(* CODESYS project Mudpi.library
   Company: ESO
   DefaultNamespace: ESO.MUDPI
   Title: ESO MUDPI Library
   Description: This library provides functionality to pack/unpack frames in the MUDPI format (Multicast UDP interface). The data format for MUDPI is described in the document "ESO-302020 - MUDPI Format".
   Placeholder: ESO MUDPI Library
   Author: Jakob Sagatowski
   Version: 1.0.1.0

Project tree, tasks and I/O mapping:
  libraries: Tc2_Standard, * (Beckhoff Automation GmbH); Tc2_System, * (Beckhoff Automation GmbH); Tc2_Utilities, * (Beckhoff Automation GmbH); Tc3_Module, * (Beckhoff Automation GmbH); TcUnit, * (www.tcunit.org)
  DUTs/
    data type ST_MudpiDataType
    data type ST_MudpiHeaderType
  GVLs/
    global variables GVL
  POUs/
    function block FB_MudpiPacket [ST]: CalculateChecksum, Data, FB_init, GetApplicationTag, GetChecksum, GetComponentId, GetFrameId, GetMaxPayloadSize, GetNumFrames, GetPayload, GetPayloadSize, GetSampleId, GetTimestamp, GetTopicId, GetVersion, IncreaseSampleId, Initialize, SetApplicationTag, SetChecksum, SetComponentId, SetFrameId, SetNumFrames, SetPayload, SetPayloadSize, SetSampleId, SetTimestamp, SetTopicId, SetVersion, Size, VerifyChecksum, VerifyPacket
  Test/
    function block FB_MudpiPacket_Test [ST]: TestChecksumCalculation, TestChecksumCalculationForPayload, TestCorrectSizeOfMudpiPacketWithAndWithoutPayload, TestPacketIntegrityMethod, TestPayloadDataSize, TestSampleIdIncreaseCorrectly, TestSerializationOfMudpiPacket, TestSetAndGetMethodForTimestamp, TestStoreAndRetrieveOfConstructorValues, TestValidAndInvalidMudpiPacketInitialization
    program PRG_TEST [ST]
  Version/
    global variables Global_Version
  VISUs/
*)

// DUTs/ST_MudpiDataType
{attribute 'pack_mode' := '1'} 
TYPE ST_MudpiDataType :
STRUCT
    header : ST_MudpiHeaderType;
    data : ARRAY[0..(GVL.MUDPI_PAYLOAD_SIZE - 1)] OF BYTE;
END_STRUCT
END_TYPE

// DUTs/ST_MudpiHeaderType
(**
 * TYPEDEF for a MUDPI header. The structure is as follows:
 *
 * UDINT TopicId         // Unique identifier of data topic
 * UINT  ComponentId     // Unique identifier of the sender
 * UINT  ApplicationTag  // For application use (not used by MUDPI)
 * UINT  Reserved1       // Reserved for future use
 * UINT  Version         // MUDPI version identifier
 * UDINT SampleId        // Rolling sample identifier (thus not unique, rather an incrementing number), incremented for each new sample
 * ULINT Timestamp       // Seconds since UNIX Epoch, following TAI time line
 * UINT  FrameId         // Frame counter for multi‐frame transmissions (starting from 1)
 * UINT  NumFrames       // Number of frames in a multi‐part message
 * UINT  PayloadSize     // Size in bytes of the payload
 * UINT  Reserved2       // Reserved for future use
 *)
 
{attribute 'pack_mode' := '1'} 
TYPE ST_MudpiHeaderType :
STRUCT
    topicId : UDINT;
    componentId : UINT;
    applicationTag : UINT;
    reserved1 : UINT;
    version : UINT;
    sampleId : UDINT;
    timestamp : ULINT;
    frameId : UINT;
    numFrames : UINT;
    payloadSize : UINT;
    reserved2 : UINT;
END_STRUCT
END_TYPE

// GVLs/GVL
(*
    MUDPI constants
*)
 
{attribute 'qualified_only'}
VAR_GLOBAL CONSTANT
    IEEE802_3_PAYLOAD_SIZE : UINT := 1500; (* = IEEE802.3 ethernet basic frame payload *)
    IPV4_HEADER_SIZE : UINT := 20;
    UDP_HEADER_SIZE : UINT := 8;
    MUDPI_PAYLOAD_SIZE : UINT := IEEE802_3_PAYLOAD_SIZE - IPV4_HEADER_SIZE - UDP_HEADER_SIZE  - SIZEOF(ST_MudpiHeaderType);
    MUDPI_VERSION : UINT := 1;
END_VAR

// Version/Global_Version
{attribute 'TcGenerated'}
{attribute 'no-analysis'}
{attribute 'linkalways'}
// This function has been automatically generated from the project information.
VAR_GLOBAL CONSTANT
	{attribute 'const_non_replaced'}
	stLibVersion_ESO_MUDPI_Library : ST_LibVersion := (iMajor := 1, iMinor := 0, iBuild := 1, iRevision := 0, sVersion := '1.0.1.0');
END_VAR

// POUs/FB_MudpiPacket
(*
    This function block gives a definition of a MUDPI packet. The MUDPI format is described in ESO document
    ESO-302020.

    As it's not possible to have more than one "constructor" in IEC61131-3, the packet is initialized in a different
    way depending on whether it's going to be used for transmission or reception.
    For transmission:
    - Just create an instance of the function block by supplying the necessary parameters to the constructor.
      All the other variables can be changed by the applicable set-methods.
    For reception:
    - Create an instance of the function block by supplying the necessary parameters to the constructor. The parameters
      can be dummy as these are going to be overwritten. Once the object is instantiated, call the method
      Initialize() on it and supply the input parameters for the data.
*)
FUNCTION_BLOCK FB_MudpiPacket
VAR
    mData : ST_MudpiDataType;
END_VAR

(*
    Calculates 16-bit UDP checksum (zero indicates no checksum).

    All 16-bit words are summed using one's complement arithmetic. Add the 16-bit values up. Each time a
    carry-out (17th bit) is produced, swing that bit around and add it back into the least significant bit.
    The sum is then one's complemented to yield the value of the UDP checksum field. If the computed
    checksum is zero, it is transmitted as all ones (the equivalent in one's complement arithmetic).
    An all zero transmitted checksum value means that the transmitter generated no checksum (for debugging
    or for higher level protocols that don't care).

*)
METHOD PUBLIC CalculateChecksum : UINT
VAR
    packetSize : UINT;
    dataPointer : POINTER TO UINT;
    dataPointerSmall : POINTER TO USINT;

    sum : UDINT := 0;
    returnValue : UINT;
END_VAR
packetSize := GetPayloadSize();
packetSize := packetSize + SIZEOF(ST_MudpiHeaderType);

dataPointer := ADR(mData.header);

// Calculate 1's complement sum of the data
WHILE (packetSize > 1) DO
    sum := sum + dataPointer^;
    dataPointer := dataPointer + SIZEOF(UINT);

    IF ((sum AND 16#80000000) = 10#1) THEN
        sum := (sum AND 16#FFFF) + (SHR(sum, 16));
    END_IF
    packetSize := packetSize - SIZEOF(UINT);
END_WHILE

IF ((packetSize AND 10#1) <> 10#0) THEN
    dataPointerSmall := dataPointer;
    sum := sum + dataPointerSmall^;
END_IF

// Add carry-over
WHILE (SHR(sum, 16)) > 10#0 DO
    sum := (sum AND 16#FFFF) + (SHR(sum, 16));
END_WHILE
returnValue := UDINT_TO_UINT(NOT sum);

IF returnValue = 0 THEN
    returnValue := NOT returnValue;
END_IF

CalculateChecksum := returnValue;
END_METHOD

(*
    Returns a pointer to the packet, be aware that the contents are big-endian!
*)
METHOD PUBLIC Data : POINTER TO BYTE
VAR
    checksum : UINT;
END_VAR
checksum := CalculateChecksum();
SetChecksum(checksum := checksum);

Data := ADR(mData);
END_METHOD

METHOD FB_init : BOOL
VAR_INPUT
    bInitRetains : BOOL; // if TRUE, the retain variables are initialized (warm start / cold start)
    bInCopyCode : BOOL;  // if TRUE, the instance afterwards gets moved into the copy code (online change)
    topicId : UDINT;
    componentId : UINT;
END_VAR
SetVersion(Version := GVL.MUDPI_VERSION);
SetFrameId(FrameId := 1);
SetNumFrames(NumFrames := 1);
SetTopicId(TopicId := topicId);
SetComponentId(ComponentId := componentId);
END_METHOD

METHOD PUBLIC GetApplicationTag : UINT
GetApplicationTag := WORD_TO_UINT(Tc2_Utilities.BE16_TO_HOST(in := UINT_TO_WORD(mData.header.applicationTag)));
END_METHOD

METHOD PUBLIC GetChecksum : UINT
VAR
    payloadSize : UINT;
    checksum : UINT;
END_VAR
payloadSize := GetPayloadSize();
Tc2_System.MEMCPY(destAddr := ADR(checksum), srcAddr := ADR(mData.data[payloadSize]), n := SIZEOF(UINT));
GetChecksum := checksum;
END_METHOD

METHOD PUBLIC GetComponentId : UINT
GetComponentId := WORD_TO_UINT(Tc2_Utilities.BE16_TO_HOST(in := UINT_TO_WORD(mData.header.componentId)));
END_METHOD

METHOD PUBLIC GetFrameId : UINT
GetFrameId := WORD_TO_UINT(Tc2_Utilities.BE16_TO_HOST(in := UINT_TO_WORD(mData.header.frameId)));
END_METHOD

(*
    Returns maximum payload size.
*)
METHOD PUBLIC GetMaxPayloadSize : UINT
GetMaxPayloadSize := GVL.MUDPI_PAYLOAD_SIZE;
END_METHOD

METHOD PUBLIC GetNumFrames : UINT
GetNumFrames := WORD_TO_UINT(Tc2_Utilities.BE16_TO_HOST(in := UINT_TO_WORD(mData.header.numFrames)));
END_METHOD

METHOD PUBLIC GetPayload : POINTER TO BYTE
GetPayload := ADR(mData.data[0]);
END_METHOD

METHOD PUBLIC GetPayloadSize : UINT
GetPayloadSize := WORD_TO_UINT(Tc2_Utilities.BE16_TO_HOST(in := UINT_TO_WORD(mData.header.payloadSize)));
END_METHOD

METHOD PUBLIC GetSampleId : UDINT
GetSampleId := DWORD_TO_UDINT(Tc2_Utilities.BE32_TO_HOST(in := UDINT_TO_DWORD(mData.header.sampleId)));
END_METHOD

(*
    This method returns the timestamp of a MUDPI packet.
    The timestamp is in seconds since UNIX Epoch, following TAI time line.
 *)
METHOD PUBLIC GetTimestamp : LREAL
VAR
    timestampLocal : LREAL;
    tmp : ULINT;
END_VAR
tmp := LWORD_TO_ULINT(Tc2_Utilities.BE64_TO_HOSTEX(in := ULINT_TO_LWORD(mdata.header.timestamp)));
Tc2_System.MEMCPY(destAddr := ADR(timestampLocal), srcAddr := ADR(tmp), n := SIZEOF(LREAL));

GetTimestamp := TimestampLocal;
END_METHOD

METHOD PUBLIC GetTopicId : UDINT
GetTopicId := DWORD_TO_UDINT(Tc2_Utilities.BE32_TO_HOST(in := UDINT_TO_DWORD(mData.header.topicId)));
END_METHOD

METHOD PUBLIC GetVersion : UINT
GetVersion := WORD_TO_UINT(Tc2_Utilities.BE16_TO_HOST(in := UINT_TO_WORD(mData.header.version)));
END_METHOD

(*
    This method increases the sample ID of the MUDPI packet.
*)
METHOD PUBLIC IncreaseSampleId
VAR
    mySampleId : UDINT;
END_VAR
mySampleId := GetSampleId();
mySampleId := mySampleId + 1;
SetSampleId(SampleId := mySampleId);
END_METHOD

(*
    This method create the MUDPI structure from a stream of bytes.
    TRUE = Creation successful, FALSE = Input data too large for MUDPI packet
*)
METHOD PUBLIC Initialize : BOOL
VAR_INPUT
    inputData : POINTER TO BYTE;
    size : UINT;
END_VAR
VAR
    sizeTmp : UINT;
END_VAR
sizeTmp := GVL.MUDPI_PAYLOAD_SIZE + SIZEOF(ST_MudpiHeaderType);

IF (size <= sizeTmp) THEN
    Tc2_System.MEMCPY(destAddr := ADR(mData), srcAddr := inputData, n := size);
    Initialize := TRUE;
ELSE
    Initialize := FALSE;
END_IF
END_METHOD

METHOD PUBLIC SetApplicationTag
VAR_INPUT
    ApplicationTag : UINT;
END_VAR
mData.header.applicationTag := WORD_TO_UINT(Tc2_Utilities.HOST_TO_BE16(in := UINT_TO_WORD(ApplicationTag)));
END_METHOD

METHOD PUBLIC SetChecksum
VAR_INPUT
    checksum : UINT;
END_VAR
VAR
    payloadSize : UINT;
END_VAR
payloadSize := GetPayloadSize();
Tc2_System.MEMCPY(destAddr := ADR(mData.data[payloadSize]), srcAddr := ADR(checksum), SIZEOF(checksum));
END_METHOD

METHOD PUBLIC SetComponentId
VAR_INPUT
    ComponentId : UINT;
END_VAR
mData.header.componentId := WORD_TO_UINT(Tc2_Utilities.HOST_TO_BE16(in := UINT_TO_WORD(ComponentId)));
END_METHOD

METHOD PUBLIC SetFrameId
VAR_INPUT
    FrameId : UINT;
END_VAR
mData.header.frameId := WORD_TO_UINT(Tc2_Utilities.HOST_TO_BE16(in := UINT_TO_WORD(FrameId)));
END_METHOD

METHOD PUBLIC SetNumFrames
VAR_INPUT
    NumFrames : UINT;
END_VAR
mData.header.numFrames := WORD_TO_UINT(Tc2_Utilities.HOST_TO_BE16(in := UINT_TO_WORD(NumFrames)));
END_METHOD

(*
    This method sets the payload of a MUDPI packet.

    payload: Pointer to any data.
    payloadSize: Size of payload data in bytes.

    Return value: TRUE = Payload set successfully, FALSE = Not possible to set payload. Payload too large for MUDPI packet.
 *)
METHOD PUBLIC SetPayload : BOOL
VAR_INPUT
    payload : POINTER TO BYTE;
    payloadSize : UINT;
END_VAR
IF (payloadSize > (GVL.MUDPI_PAYLOAD_SIZE - SIZEOF(UINT))) THEN // SIZEOF(UINT) = Checksum
    SetPayload := FALSE;
ELSE
    IF (payloadSize > 0) THEN
        SetPayloadSize(payloadSize);
        Tc2_System.MEMCPY(destAddr := ADR(mData.data[0]), srcAddr := payload, n := payloadSize);
    END_IF
    SetPayload := TRUE;
END_IF
END_METHOD

METHOD PUBLIC SetPayloadSize
VAR_INPUT
    PayloadSize : UINT;
END_VAR
mData.header.payloadSize := WORD_TO_UINT(Tc2_Utilities.HOST_TO_BE16(in := UINT_TO_WORD(PayloadSize)));
END_METHOD

METHOD PUBLIC SetSampleId
VAR_INPUT
    SampleId : UDINT;
END_VAR
mData.header.sampleId := DWORD_TO_UDINT(Tc2_Utilities.HOST_TO_BE32(in := UDINT_TO_DWORD(SampleId)));
END_METHOD

(*
    This method sets the timestamp of a MUDPI packet.
    The timestamp is in seconds since UNIX Epoch, following TAI time line.
 *)
METHOD PUBLIC SetTimestamp
VAR_INPUT
    Timestamp : LREAL;
END_VAR
VAR
    TimestampLocal : ULINT;
END_VAR
Tc2_System.MEMCPY(destAddr := ADR(TimestampLocal), srcAddr := ADR(Timestamp), n := SIZEOF(LREAL));
mData.header.timestamp := LWORD_TO_ULINT(Tc2_Utilities.HOST_TO_BE64EX(in := ULINT_TO_LWORD(TimestampLocal)));
END_METHOD

METHOD PUBLIC SetTopicId
VAR_INPUT
    TopicId : UDINT;
END_VAR
mData.header.topicId := DWORD_TO_UDINT(Tc2_Utilities.HOST_TO_BE32(in := UDINT_TO_DWORD(TopicId)));
END_METHOD

METHOD PUBLIC SetVersion
VAR_INPUT
    Version : UINT;
END_VAR
mData.header.version := WORD_TO_UINT(Tc2_Utilities.HOST_TO_BE16(in := UINT_TO_WORD(Version)));
END_METHOD

(*
    This method returns the size of the MUDPI packet in bytes.
    The return value is the size of the packet in bytes, i.e. MUDPI header + payload + checksum.
 *)
METHOD PUBLIC Size : UINT
VAR
    payloadSize : UINT;
    sizeOfMudpiHeader : UINT := SIZEOF(ST_MudpiHeaderType);
    sizeOfChecksum : UINT := SIZEOF(UINT);
END_VAR
payloadSize := GetPayloadSize();
Size := payloadSize + sizeOfMudpiHeader + sizeOfChecksum;
END_METHOD

(*
    This method verifies, if the checksum of a MUDPI packet is correct.
    TRUE = Checksum does match the content of the packet, FALSE = checksum does not match.
*)
METHOD PUBLIC VerifyChecksum : BOOL
VAR
    checksum1 : UINT;
    checksum2 : UINT;
END_VAR
checksum1 := GetChecksum();
checksum2 := CalculateChecksum();

// The MUDPI standard allows to omit the checksum calculation
IF ((checksum1 = 0) OR (checksum2 = 0)) THEN
    VerifyChecksum := TRUE;
ELSE
    VerifyChecksum := (checksum1 = checksum2);
END_IF
END_METHOD

(*
    This method verifies, if the internal structure of a MUDPI packet is correct.
    TRUE = internal structure of packet is correct, FALSE = internal structure of packet is not correct
*)
METHOD PUBLIC VerifyPacket : BOOL
VAR
    version : UINT;
    frameId : UINT;
    numFrames : UINT;
    topicId : UDINT;
    componentId : UINT;
    checksumCorrect : BOOL;
    packetCorrect : BOOL;
END_VAR
version := GetVersion();
frameId := GetFrameId();
numFrames := GetNumFrames();
topicId := GetTopicId();
componentId := GetComponentId();

checksumCorrect := VerifyChecksum();
packetCorrect := (version = GVL.MUDPI_VERSION) AND (frameId <= numFrames) AND (topicId <> 0) AND (componentId <> 0);

VerifyPacket := (checksumCorrect AND packetCorrect);
END_METHOD

END_FUNCTION_BLOCK

// Test/FB_MudpiPacket_Test
(*
    This is the test-FB for FB_MudpiPacket
*)
{attribute 'call_after_init'}
FUNCTION_BLOCK FB_MudpiPacket_Test EXTENDS TcUnit.FB_TestSuite
VAR CONSTANT
    cTopicId : UDINT := 10;
    cComponentId : UINT := 500;
END_VAR

TestStoreAndRetrieveOfConstructorValues();
TestCorrectSizeOfMudpiPacketWithAndWithoutPayload();
TestPayloadDataSize();
TestChecksumCalculationForPayload();
TestSampleIdIncreaseCorrectly();
TestPacketIntegrityMethod();
TestSerializationOfMudpiPacket();
TestValidAndInvalidMudpiPacketInitialization();
TestSetAndGetMethodForTimestamp();
TestChecksumCalculation();

(*
    Test checksum calculation for given header

    The header should be according to:
    - TopicId = 500
    - ComponentId = 10
    - ApplicationTag = 300
    - SampleId = 422
    - NumFrames = 212
    - Version = 1
    - Timestamp = 0
    - FrameId = 1
    - No Payload
*)
METHOD PRIVATE TestChecksumCalculation
VAR
    // Construct MUDPI packet
    packet : FB_MudpiPacket(topicId := 500, componentId := 10);

    checksum : UINT;
END_VAR
TEST('TestChecksumCalculation');

packet.SetApplicationTag(ApplicationTag := 300);
packet.SetSampleId(SampleId := 422);
packet.SetNumFrames(NumFrames := 212);
packet.SetVersion(Version := 1);
packet.SetTimeStamp(Timestamp := 0.0);
packet.SetFrameId(FrameId := 1);

checksum := packet.CalculateChecksum();

AssertEquals_UINT(Expected := Tc2_Utilities.HOST_TO_BE16(16#FA59),
                  Actual := checksum,
                  Message := 'Calculated checksum is not correct');

TEST_FINISHED();
END_METHOD

(*
    Test checksum calculation for a given payload, and for empty payload data.
*)
METHOD PRIVATE TestChecksumCalculationForPayload
VAR
    // Construct MUDPI packet
    packet : FB_MudpiPacket(topicId := cTopicId, componentId := cComponentId);

    payloadParam : STRING := 'This is a payload';
    checkChecksum1 : BOOL;

    checksum1 : UINT;
    checksum2 : UINT;
END_VAR
TEST('TestChecksumCalculationForPayload');

packet.SetPayload(payload := ADR(payloadParam),
                  payloadSize := SIZEOF(payloadParam));

// Invoke calculation of checksum
packet.Data();

// Verify, if checksum was calculated correctly
checkChecksum1 := packet.VerifyChecksum();

AssertTrue(Condition := checkChecksum1,
           Message := 'Checksum not calculated correctly');

// Calculate checksum, and verify if identical to setting in MUDPI packet
checksum1 := packet.CalculateChecksum();
checksum2 := packet.GetChecksum();

AssertEquals_UINT(Expected := checksum1,
                  Actual := checksum2,
                  Message := 'Calculated checksum not identical with the one in MUDPI packet');

TEST_FINISHED();
END_METHOD

(*
    Test correct return value of size() method with and without payload.
    Test correct return value of getMaxPayloadSize
*)
METHOD PRIVATE TestCorrectSizeOfMudpiPacketWithAndWithoutPayload
VAR
    // Construct MUDPI packet
    packet : FB_MudpiPacket(topicId := cTopicId, componentId := cComponentId);

    sizeHeader : UINT;
    sizeReturned : UINT;
    sizeCorrect : BOOL;

    payloadSize : UINT;
    maxPayloadSize : UINT;

    payload : STRING(9) := '123456789'; // 10 bytes (including the null-character)
END_VAR
TEST('TestCorrectSizeOfMudpiPacketWithAndWithoutPayload');

// Test correct size of MUDPI header
sizeHeader := SIZEOF(ST_MudpiHeaderType);
sizeReturned := packet.Size() - SIZEOF(UINT); // Checksum

AssertEquals_UINT(Expected := sizeHeader,
                  Actual := sizeReturned,
                  Message := 'Size of MUDPI header not correct');

// Test correct size of MUDPI packet with payload of 10 bytes (+checksum internally)
packet.SetPayload(payload := ADR(payload),
                  payloadSize := SIZEOF(payload));
payloadSize := packet.GetPayloadSize();
sizeReturned := packet.Size();
AssertEquals_UINT(Expected := SIZEOF(payload),
                  Actual := payloadSize,
                  Message := 'Size of MUDPI payload not correct');
AssertEquals_UINT(Expected := (sizeHeader + SIZEOF(payload) + SIZEOF(UINT)), // SIZEOF(UINT) = Checksum
                  Actual := sizeReturned,
                  Message := 'Total size of MUDPI-packet including payload not correct');

// Test correct return value of getMaxPayloadSize
maxPayloadSize := packet.GetMaxPayloadSize();
AssertEquals_UINT(Expected := GVL.MUDPI_PAYLOAD_SIZE,
                  Actual := maxPayloadSize,
                  Message := 'The returned value for maximum payload size for the MUDPI packet is not correct');

TEST_FINISHED();
END_METHOD

METHOD PRIVATE TestPacketIntegrityMethod
VAR
    // Construct MUDPI packet
    packet : FB_MudpiPacket(topicId := cTopicId, componentId := cComponentId);
END_VAR
TEST('TestPacketIntegrityMethod');

packet.IncreaseSampleId();

AssertTrue(Condition := packet.VerifyPacket(),
           Message := 'MUDPI packet integrity failed');

TEST_FINISHED();
END_METHOD

(*
    Test setting and retrieving of payload data.
    Test the correct return value for the payload length for packets with and without payload data.
*)
METHOD PRIVATE TestPayloadDataSize
VAR
    // Construct MUDPI packet
    packet : FB_MudpiPacket(topicId := cTopicId, componentId := cComponentId);

    emptyPayloadSize : UINT;
    newPayloadSize : UINT;

    payload : STRING(17) := 'This is a payload'; // 18 bytes (including the null-character)
END_VAR
TEST('TestPayloadDataSize');

// Verify that the payload is empty
emptyPayloadSize := packet.GetPayloadSize();

AssertEquals_UDINT(Expected := 0,
                   Actual := emptyPayloadSize,
                   Message := 'MUDPI payload size is not zero');

// Set a new payload, and verify correct length
packet.SetPayload(payload := ADR(payload),
                  payloadSize := SIZEOF(payload));

newPayloadSize := packet.GetPayloadSize();

AssertEquals_UDINT(Expected := SIZEOF(payload),
                   Actual := newPayloadSize,
                   Message := 'MUDPI payload size is not correct');

TEST_FINISHED();
END_METHOD

(*
    Test, if the sampleId is increased correctly.
*)
METHOD TestSampleIdIncreaseCorrectly
VAR
    // Construct MUDPI packet
    packet : FB_MudpiPacket(topicId := cTopicId, componentId := cComponentId);

    firstSampleId : UDINT;
    secondSampleId : UDINT;
END_VAR
TEST('TestSampleIdIncreaseCorrectly');

// Get initial and increased sampleId
firstSampleId := packet.GetSampleId();
packet.IncreaseSampleId();
secondSampleId := packet.GetSampleId();

AssertEquals_UDINT(Expected := 0,
                   Actual := firstSampleId,
                   Message := 'First Sample-ID not correct');

AssertEquals_UDINT(Expected := 1,
                   Actual := secondSampleId,
                   Message := 'Second Sample-ID not correct');

TEST_FINISHED();
END_METHOD

(*
    Test correct serialization of the MUDPI packet.
*)
METHOD PRIVATE TestSerializationOfMudpiPacket
VAR
    // Construct MUDPI packet
    packet : FB_MudpiPacket(topicId := cTopicId, componentId := cComponentId);

    aByteArray : ARRAY[0..3] OF BYTE;
    serializedData : POINTER TO BYTE;
END_VAR
TEST('TestSerializationOfMudpiPacket');

(* We expect big-endian format, i.e. the bytes in the following order:
    Topic-ID: 0x11, 0x22, 0x33, 0x44
    Component-ID: 0x55, 0x66
    Application-tag: 0x77, 0x88
    Reserved: 0x00, 0x00
    Version: 0x99, 0xAA
    Sample-ID: 0xBB, 0xCC, 0xDD, 0xEE
    Timestamp: 0x40, 0x93, 0x4A, 0x00, 0x00, 0x00, 0x00, 0x00
    Frame-ID: 0x88, 0x99
    NumFrames: 0xAA, 0xBB
    Payload size: 0x01, 0xFF
    Reserved: 0x00, 0x00
*)
packet.SetTopicId(16#11223344);
packet.SetComponentId(16#5566);
packet.SetApplicationTag(16#7788);
packet.SetVersion(16#99AA);
packet.SetSampleId(16#BBCCDDEE);
packet.SetTimeStamp(1234.5); // 1234.5 = 16#40934A0000000000
packet.SetFrameId(16#8899);
packet.SetNumFrames(16#AABB);
packet.SetPayloadSize(16#01FF);

serializedData := packet.Data();
AssertEquals_BYTE(Expected := 16#11,
                  Actual := serializedData[0],
                  Message := 'Byte 0 is not correctly serialized');
AssertEquals_BYTE(Expected := 16#22,
                  Actual := serializedData[1],
                  Message := 'Byte 1 is not correctly serialized');
AssertEquals_BYTE(Expected := 16#33,
                  Actual := serializedData[2],
                  Message := 'Byte 2 is not correctly serialized');
AssertEquals_BYTE(Expected := 16#44,
                  Actual := serializedData[3],
                  Message := 'Byte 3 is not correctly serialized');
AssertEquals_BYTE(Expected := 16#55,
                  Actual := serializedData[4],
                  Message := 'Byte 4 is not correctly serialized');
AssertEquals_BYTE(Expected := 16#66,
                  Actual := serializedData[5],
                  Message := 'Byte 5 is not correctly serialized');
AssertEquals_BYTE(Expected := 16#77,
                  Actual := serializedData[6],
                  Message := 'Byte 6 is not correctly serialized');
AssertEquals_BYTE(Expected := 16#88,
                  Actual := serializedData[7],
                  Message := 'Byte 7 is not correctly serialized');
AssertEquals_BYTE(Expected := 16#00,
                  Actual := serializedData[8],
                  Message := 'Byte 8 is not correctly serialized');
AssertEquals_BYTE(Expected := 16#00,
                  Actual := serializedData[9],
                  Message := 'Byte 9 is not correctly serialized');
AssertEquals_BYTE(Expected := 16#99,
                  Actual := serializedData[10],
                  Message := 'Byte 10 is not correctly serialized');
AssertEquals_BYTE(Expected := 16#AA,
                  Actual := serializedData[11],
                  Message := 'Byte 11 is not correctly serialized');
AssertEquals_BYTE(Expected := 16#BB,
                  Actual := serializedData[12],
                  Message := 'Byte 12 is not correctly serialized');
AssertEquals_BYTE(Expected := 16#CC,
                  Actual := serializedData[13],
                  Message := 'Byte 13 is not correctly serialized');
AssertEquals_BYTE(Expected := 16#DD,
                  Actual := serializedData[14],
                  Message := 'Byte 14 is not correctly serialized');
AssertEquals_BYTE(Expected := 16#EE,
                  Actual := serializedData[15],
                  Message := 'Byte 15 is not correctly serialized');

AssertEquals_BYTE(Expected := 16#40,
                  Actual := serializedData[16],
                  Message := 'Byte 16 is not correctly serialized');
AssertEquals_BYTE(Expected := 16#93,
                  Actual := serializedData[17],
                  Message := 'Byte 17 is not correctly serialized');
AssertEquals_BYTE(Expected := 16#4A,
                  Actual := serializedData[18],
                  Message := 'Byte 18 is not correctly serialized');
AssertEquals_BYTE(Expected := 16#00,
                  Actual := serializedData[19],
                  Message := 'Byte 19 is not correctly serialized');
AssertEquals_BYTE(Expected := 16#00,
                  Actual := serializedData[20],
                  Message := 'Byte 20 is not correctly serialized');
AssertEquals_BYTE(Expected := 16#00,
                  Actual := serializedData[21],
                  Message := 'Byte 21 is not correctly serialized');
AssertEquals_BYTE(Expected := 16#00,
                  Actual := serializedData[22],
                  Message := 'Byte 22 is not correctly serialized');
AssertEquals_BYTE(Expected := 16#00,
                  Actual := serializedData[23],
                  Message := 'Byte 23 is not correctly serialized');

AssertEquals_BYTE(Expected := 16#88,
                  Actual := serializedData[24],
                  Message := 'Byte 24 is not correctly serialized');
AssertEquals_BYTE(Expected := 16#99,
                  Actual := serializedData[25],
                  Message := 'Byte 25 is not correctly serialized');
AssertEquals_BYTE(Expected := 16#AA,
                  Actual := serializedData[26],
                  Message := 'Byte 26 is not correctly serialized');
AssertEquals_BYTE(Expected := 16#BB,
                  Actual := serializedData[27],
                  Message := 'Byte 27 is not correctly serialized');
AssertEquals_BYTE(Expected := 16#01,
                  Actual := serializedData[28],
                  Message := 'Byte 28 is not correctly serialized');
AssertEquals_BYTE(Expected := 16#FF,
                  Actual := serializedData[29],
                  Message := 'Byte 29 is not correctly serialized');
AssertEquals_BYTE(Expected := 16#00,
                  Actual := serializedData[30],
                  Message := 'Byte 30 is not correctly serialized');
AssertEquals_BYTE(Expected := 16#00,
                  Actual := serializedData[31],
                  Message := 'Byte 31 is not correctly serialized');

TEST_FINISHED();
END_METHOD

(*
    Test set() and get() methods for the timestamp LREAL value.
*)
METHOD PRIVATE TestSetAndGetMethodForTimestamp
VAR
    // Construct MUDPI packet
    packet : FB_MudpiPacket(topicId := cTopicId, componentId := cComponentId);

    timestamp1 : LREAL := 1234.5;
    timestamp2 : LREAL;
END_VAR
TEST('TestSetAndGetMethodForTimestamp');

packet.SetTimeStamp(Timestamp := timestamp1);
timestamp2 := packet.GetTimestamp();

AssertEquals_LREAL(Expected := timestamp1,
                   Actual := timestamp2,
                   Delta := 0.0,
                   Message := 'Timestamps differ');

TEST_FINISHED();
END_METHOD

(*
    Test constructor of a MUDPI packet with topicId and componentId.
    Test, if topicId and componentId are correctly stored and retrieved.
    Test, if MUDPI-version is correctly stored.
    Test, if frame identity and number of frames is correctly stored and retrieved
*)
METHOD PRIVATE TestStoreAndRetrieveOfConstructorValues
VAR
    // Construct MUDPI packet
    packet : FB_MudpiPacket(topicId := cTopicId, componentId := cComponentId);

    topicId : UDINT;
    componentId : UINT;
    version : UINT;
    frameId : UINT;
    numFrames : UINT;
END_VAR
TEST('TestStoreAndRetrieveOfConstructorValues');

// Retrieve topicId and componentId, compare with constructed values
topicId := packet.GetTopicId();
componentId := packet.GetComponentId();

AssertEquals_UDINT(Expected := cTopicId,
                   Actual := topicId,
                   Message := 'Not correct $'Topic-ID$' retrieved');

AssertEquals_UINT(Expected := cComponentId,
                  Actual := componentId,
                  Message := 'Not correct $'Component-ID$' retrieved');

// Test MUDPI version, frameId, and numFrames
version := packet.GetVersion();
frameId := packet.GetFrameId();
numFrames := packet.GetNumFrames();

AssertEquals_UINT(Expected := GVL.MUDPI_VERSION,
                  Actual := version,
                  Message := 'Not correct $'version$' retrieved');

AssertEquals_UINT(Expected := 1,
                  Actual := frameId,
                  Message := 'Not correct $'Frame-ID$' retrieved');

AssertEquals_UINT(Expected := 1,
                  Actual := numFrames,
                  Message := 'Not correct $'NumberOfFrames$' retrieved');

TEST_FINISHED();
END_METHOD

(*
    Test valid and invalid MUDPI packet size initialization
*)
METHOD TestValidAndInvalidMudpiPacketInitialization
VAR
    // Construct MUDPI packet
    packet : FB_MudpiPacket(topicId := cTopicId, componentId := cComponentId);

    sizeOk : STRING(99) := ''; // 100 bytes (incl. null-character)
    sizeNotOk : STRING(GVL.IEEE802_3_PAYLOAD_SIZE+9) := ''; // 1510 bytes (incl. null-character)

    bResultOfInitialization : BOOL;
END_VAR
TEST('TestValidAndInvalidMudpiPacketInitialization');

// Valid initialization
bResultOfInitialization := packet.Initialize(inputData := ADR(sizeOk),
                                             size := SIZEOF(sizeOk));

AssertTrue(Condition := bResultOfInitialization,
           Message := 'Failed to initialize MUDPI packet');

// Non-valid initialization
bResultOfInitialization := packet.Initialize(inputData := ADR(sizeNotOk),
                                             size := SIZEOF(sizeNotOk));

AssertFalse(Condition := bResultOfInitialization,
            Message := 'Initialized MUDPI packet even though the size is too big');

TEST_FINISHED();
END_METHOD

END_FUNCTION_BLOCK

// Test/PRG_TEST
(*
    This is the main program for execution of the unit tests.
*)
PROGRAM PRG_TEST
VAR
    (* Test function blocks *)
    fbMudpiPacket_Test : FB_MudpiPacket_Test;
END_VAR

TcUnit.RUN();

END_PROGRAM
